(*
	Function Block which performs a bang-bang control loop.
*)
{attribute 'OPC.UA.DA.StructuredType' := '1'}
FUNCTION_BLOCK FB_BangBangControl_Analog EXTENDS FB_BaseDevice
VAR_INPUT PERSISTENT
	{attribute 'OPC.UA.DA' := '1'}
	rAlarmHigh : REAL;
	{attribute 'OPC.UA.DA' := '1'}
	rAlarmLow : REAL;
	{attribute 'OPC.UA.DA' := '1'}
	rLimitHigh : REAL; // the upper limit of the desirable range (when the downward adjustment is activated)
	{attribute 'OPC.UA.DA' := '1'}
	rLimitLow : REAL; // lower limit of the desirable range (when the upward adjustment is activated)
	{attribute 'OPC.UA.DA' := '1'}
	nAdjustDelay : INT := 30; // min time in seconds between adjustments
	{attribute 'OPC.UA.DA' := '1'}
	nAdjustDownIncrement : REAL := 0.5;
	{attribute 'OPC.UA.DA' := '1'}
	nAdjustUpIncrement : REAL := 0.5; 
	{attribute 'OPC.UA.DA' := '1'}
	rCurrentValue : REAL; 
	{attribute 'OPC.UA.DA' := '1'}
	bEnabled : BOOL; 
	{attribute 'OPC.UA.DA' := '1'}
	sParameterName : STRING;
	
	{attribute 'OPC.UA.DA' := '1'}
	nControlValue: POINTER TO REAL;
	{attribute 'OPC.UA.DA' := '1'}
	nControlValueCopy: REAL;
	
	{attribute 'OPC.UA.DA' := '1'}
	Mode:    E_CTRL_MODE;
END_VAR

VAR_OUTPUT

	{attribute 'OPC.UA.DA' := '1'}
	bAlarmHigh : BOOL;
	{attribute 'OPC.UA.DA' := '1'}
	bAlarmLow : BOOL;
END_VAR

VAR
	tAdjustDownTimer : TON;
	tAdjustUpTimer : TON;
	tAdjustDelayTimer : TON;
	bAdjustDownActive : BOOL;
	bAdjustUpActive : BOOL;
	bDelayActive : BOOL;
END_VAR

IF eState = E_DeviceState.RUNNING THEN
	timers();
	// output signals
	IF bAdjustUpActive THEN
		IF NOT (nControlValue^ > ((rLimitHigh + rLimitLow)/2.0)) THEN
			nControlValue^ := nControlValue^ + nAdjustUpIncrement;
		END_IF
		bAdjustUpActive := FALSE;	
	END_IF
	
	IF bAdjustDownActive THEN
		IF NOT (nControlValue^ <= 16) THEN
			nControlValue^ := nControlValue^ - nAdjustDownIncrement;
		END_IF
		bAdjustDownActive := FALSE;	
	END_IF
	
	// alarms
	bAlarmHigh := (rCurrentValue >= rAlarmHigh);
	bAlarmLow := (rCurrentValue <= rAlarmLow);
ELSE
	bAlarmHigh := FALSE;
	bAlarmLow := FALSE;
	// clear the delay timer 
	tAdjustDelayTimer.PT := INT_TO_TIME(0);
END_IF

nControlValueCopy := nControlValue^;

METHOD setState : BOOL
VAR_INPUT
	state : E_DeviceState;
END_VAR

eState := state;
END_METHOD


(*
	Run the timers for delay, adjust up and adjust down
*)
METHOD timers : BOOL
VAR_INPUT
END_VAR
tAdjustDelayTimer(IN := bDelayActive, PT := INT_TO_TIME(nAdjustDelay) * 1000);


IF tAdjustDelayTimer.Q THEN
	// the delay timer is finished so check if we need to activate an adjustment
	
	//bAdjustDownActive := (rCurrentValue > rLimitHigh);
	//bAdjustUpActive := (rCurrentValue < rLimitLow);
	
	bAdjustDownActive := (rCurrentValue > ((rLimitHigh + rLimitLow)/2.0)+0.6);
	bAdjustUpActive := (rCurrentValue < ((rLimitHigh + rLimitLow)/2.0)-0.6);
	
END_IF

// run the delay timer whenever we are not activating an output
bDelayActive := NOT bAdjustDownActive AND NOT bAdjustUpActive;
END_METHOD

END_FUNCTION_BLOCK

(* stored: Version 1.1.0.1, ProductVersion 3.1.4024.12
   POU FB_BangBangControl_Analog: Id {0d66fff2-b416-4a31-af59-59956e6c5d2e}, SpecialFunc None
   Method setState: Id {8817253c-2009-4706-a0ca-1319c20a4e0e}
   Method timers: Id {b9d7fc3d-e24c-4267-8bd9-0f92d0c9cf43} *)
